GLOBALCONSTANTS DefaultPool_TECU_Numeric (* Numeric object pool constants (ID, Scale, Offset, Decimals) *)
  PACKAGE Uebungen::const::UT::TECU;
  VAR_GLOBAL CONSTANT
    OutputNumber_Wheel_based_machine_speed_km_h : isobus::UT::io::NumericValue::NumericObjectPool_S := (u16ObjId := 12000, r32Scale := 0.0036, i32Offset := 0, u8Decimals := 1);
    OutputNumber_Wheel_based_machine_speed_m_s : isobus::UT::io::NumericValue::NumericObjectPool_S := (u16ObjId := 12001, r32Scale := 0.001, i32Offset := 0, u8Decimals := 1);
    OutputNumber_Ground_based_machine_speed_km_h : isobus::UT::io::NumericValue::NumericObjectPool_S := (u16ObjId := 12002, r32Scale := 0.0036, i32Offset := 0, u8Decimals := 1);
    OutputNumber_Ground_based_machine_speed_m_s : isobus::UT::io::NumericValue::NumericObjectPool_S := (u16ObjId := 12003, r32Scale := 0.001, i32Offset := 0, u8Decimals := 1);
    OutputNumber_Wheel_based_machine_distance_km : isobus::UT::io::NumericValue::NumericObjectPool_S := (u16ObjId := 12004, r32Scale := 0.000001, i32Offset := 0, u8Decimals := 1);
    OutputNumber_Wheel_based_machine_distance_m : isobus::UT::io::NumericValue::NumericObjectPool_S := (u16ObjId := 12005, r32Scale := 0.001, i32Offset := 0, u8Decimals := 1);
    OutputNumber_Rear_PTO_output_shaft_speed : isobus::UT::io::NumericValue::NumericObjectPool_S := (u16ObjId := 12006, r32Scale := 0.125, i32Offset := 0, u8Decimals := 1);
  END_VAR
END_GLOBALCONSTANTS
